// TIA Portal V19 export
DATA_BLOCK "ALARM DB PLC 2"   // DB37
{ S7_Optimized_Access := 'FALSE' }
   VAR
      "P-201 A RO 1 FEED PUMP TRIP" : Bool;
      "P-201 B RO 1 FEED PUMP TRIP" : Bool;
      "P-201 C RO 1 FEED PUMP TRIP" : Bool;
      "P-301 A RO 1 HPP PUMP TRIP" : Bool;
      "P-301 B RO B HPP PUMP TRIP" : Bool;
      "P-401 A RO 2 FEED PUMP TRIP" : Bool;
      "P-401 B RO 2 FEED PUMP TRIP" : Bool;
      "P-401 C RO 2 FEED PUMP TRIP" : Bool;
      "P 401 A RO 2 HPP PUMP TRIP" : Bool;
      "P-401 B RO 2 HPP PUMP TRIP" : Bool;
      "P-501 A EDI FEED PUMP TRIP" : Bool;
      "P-501 B EDI FEED PUMP TRIP" : Bool;
      "P-501 C EDI FEED PUMP TRIP" : Bool;
      "EDI 501 A TRIP" : Bool;
      "EDI 501 B TRIP" : Bool;
      "P-201 A RO 1 FEED PUMP_FEEDBACK FAIL" : Bool;
      "P-201 B RO 1 FEED PUMP_FEEDBACK FAIL" : Bool;
      "P-201 C RO 1 FEED PUMP_FEEDBACK FAIL" : Bool;
      "P-301 A RO 1 HPP PUMP_FEEDBACK FAIL" : Bool;
      "P-301 B RO B HPP PUMP_FEEDBACK FAIL" : Bool;
      "P-401 A RO 2 FEED PUMP_FEEDBACK FAIL" : Bool;
      "P-401 B RO 2 FEED PUMP_FEEDBACK FAIL" : Bool;
      "P-401 C RO 2 FEED PUMP_FEEDBACK FAIL" : Bool;
      "P 401 A RO 2 HPP PUMP_FEEDBACK FAIL" : Bool;
      "P-401 B RO 2 HPP PUMP_FEEDBACK FAIL" : Bool;
      "P-501 A EDI FEED PUMP_FEEDBACK FAIL" : Bool;
      "P-501 B EDI FEED PUMP_FEEDBACK FAIL" : Bool;
      "P-501 C EDI FEED PUMP_FEEDBACK FAIL" : Bool;
      "EDI 501 A _FEEDBACK FAIL" : Bool;
      "EDI 501 B_FEEDBACK FAIL" : Bool;
      "RO-01 ORP DUMP VALVE ABV-301 OPEN COMMOND FAIL" : Bool;
      "RO-01 ORP DUMP VALVE ABV-301 CLOSE COMMOND FAIL" : Bool;
      "RO-01 ORP PROCESS VALVE ABV-302 OPEN COMMOND FAIL" : Bool;
      "RO-01 ORP PROCESS VALVE ABV-302 CLOSE COMMOND FAIL" : Bool;
      "RO-1 A AUTO FLUSING VALVE AGLV-301 OPEN COMMOND FAIL" : Bool;
      "RO-1 A AUTO FLUSING VALVE AGLV-301 CLOSE COMMOND FAIL" : Bool;
      "RO-1 B AUTO FLUSING VALVE AGLV-302 OPEN COMMOND FAIL" : Bool;
      "RO-1 B AUTO FLUSING VALVE AGLV-302 CLOSE COMMOND FAIL" : Bool;
      "RO-2 A AUTO FLUSING VALVE AGLV-401 OPEN COMMOND FAIL" : Bool;
      "RO-2 A AUTO FLUSING VALVE AGLV-401 CLOSE COMMOND FAIL" : Bool;
      "RO-2 B AUTO FLUSING VALVE AGLV-402 OPEN COMMOND FAIL" : Bool;
      "RO-2 B AUTO FLUSING VALVE AGLV-402 CLOSE COMMOND FAIL" : Bool;
      "EDI AUTO DUMP VALVE ABV-501 OPEN COMMOND FAIL" : Bool;
      "EDI AUTO DUMP VALVE ABV-501 CLOSE COMMOND FAIL" : Bool;
      "DM TANK INLET VALVE ABV-502 OPEN COMMOND FAIL" : Bool;
      "DM TANK INLET VALVE ABV-502 CLOSE COMMOND FAIL" : Bool;
      "RO-02 FEED TANK LEVEL ( LT-401)- LOW LOW" : Bool;
      "RO-02 FEED TANK LEVEL ( LT-401)- HIGH HIGH" : Bool;
      "EDI FEED TANK LEVEL ( LT-501)- LOW LOW" : Bool;
      "EDI FEED TANK LEVEL ( LT-501)- HIGH HIGH" : Bool;
      "DM WATER STORAGE TANK  LEVEL ( LT-502)- LOW LOW" : Bool;
      "DM WATER STORAGE TANK LEVEL ( LT-502)- HIGH HIGH" : Bool;
      "RO-01A LPS-301 LOW" : Bool;
      "RO-01 B LPS-302 LOW" : Bool;
      "RO-01 A HPS-301 HIGH" : Bool;
      "RO-01B HPS-302 HIGH" : Bool;
      "RO-02A LPS-401 LOW" : Bool;
      "RO-02B LPS-402 LOW" : Bool;
      "RO-02A HPS-401 HIGH" : Bool;
      "RO-02 B HPS-402 HIGH" : Bool;
      "EDI-501A FEED PRESSURE PT-501 LOW" : Bool;
      "PT-501A LOW_SET VALIDATION TIME OVER_(SYSTEM STOP)" : Bool;
      "EDI-501A FEED PRESSURE PT-501 HIGH" : Bool;
      "PT-501A HIGH_SET VALIDATION TIME OVER_(SYSTEM STOP)" : Bool;
      "EDI-501B FEED PRESSURE PT-502 LOW" : Bool;
      "PT-501B LOW_SET VALIDATION TIME OVER_(SYSTEM STOP)" : Bool;
      "EDI-501B FEED PRESSURE PT-502 HIGH" : Bool;
      "PT-501B HIGH_SET VALIDATION TIME OVER_(SYSTEM STOP)" : Bool;
      "EDI-501B CONCENTRATE OUT PRESSURE PT-503 HIGH" : Bool;
      "PT-503 HIGH_SET VALIDATION TIME OVER_(SYSTEM STOP)" : Bool;
      "EDI-501A PRODUCT OUT PRESSURE PT-504 HIGH" : Bool;
      "PT-504 HIGH_SET VALIDATION TIME OVER_(SYSTEM STOP)" : Bool;
      "EDI-501A CONCENTRATE OUT PRESSURE PT-505 HIGH" : Bool;
      "PT-505 HIGH_SET VALIDATION TIME OVER_(SYSTEM STOP)" : Bool;
      "EDI-501B PRODUCT OUT PRESSURE PT-506 HIGH" : Bool;
      "PT-506 HIGH_SET VALIDATION TIME OVER_(SYSTEM STOP)" : Bool;
      "RO-01 FEED PHIT-301 HIGH" : Bool;
      "RO-01 FEED PHIT-301 LOW" : Bool;
      "RO-01 PRODUCT PHIT-302 HIGH" : Bool;
      "RO-01 PRODUCT PHIT-302 LOW" : Bool;
      "RO-02 FEED PHIT-401 HIGH" : Bool;
      "RO-02 FEED PHIT-401 LOW" : Bool;
      "RO-02 PRODUCT PHIT-402 HIGH" : Bool;
      "RO-02 PRODUCT PHIT-402 LOW" : Bool;
      "EDI-501A PRODUCT OUT  PHIT-501 HIGH" : Bool;
      "EDI-501A PRODUCT OUT  PHIT-501 LOW" : Bool;
      "EDI-501B PRODUCT OUT  PHIT-502 HIGH" : Bool;
      "EDI-501B PRODUCT OUT PHIT-502 LOW" : Bool;
      "RO-01 FEED CIT-301 HIGH" : Bool;
      "CIT-301 HIGH_SET VALIDATION TIME OVER_(SYSTEM STOP)" : Bool;
      "RO-01 PRODUCT CIT-302 HIGH" : Bool;
      "CIT-302 HIGH_SET VALIDATION TIME OVER_(SYSTEM STOP)" : Bool;
      "RO-02 FEED CIT-401 HIGH" : Bool;
      "CIT-401 HIGH_SET VALIDATION TIME OVER_(SYSTEM STOP)" : Bool;
      "RO-02 PRODUCT CIT-402 HIGH" : Bool;
      "CIT-402 HIGH_SET VALIDATION TIME OVER_(SYSTEM STOP)" : Bool;
      "EDI-501A PRODUCT OUT RIT-501 HIGH" : Bool;
      "RIT-501A HIGH_SET VALIDATION TIME OVER_(SYSTEM STOP)" : Bool;
      "EDI-501B PRODUCT OUT RIT-502 HIGH" : Bool;
      "RIT-501B HIGH_SET VALIDATION TIME OVER_(SYSTEM STOP)" : Bool;
      "ORP-301 HIGH" : Bool;
      "ORP-301 HIGH_SET VALIDATION TIME OVER_(SYSTEM STOP)" : Bool;
      "EDI-501A FEED PRESSURE FIT-501 LOW" : Bool;
      "FIT-501  LOW_SET VALIDATION TIME OVER_(SYSTEM STOP)" : Bool;
      "EDI-501B FEED PRESSURE FIT-502 LOW" : Bool;
      "FIT-501 LOW_SET VALIDATION TIME OVER_(SYSTEM STOP)" : Bool;
      "EDI-501B CONCENTRATE OUT PRESSURE FIT-503 LOW" : Bool;
      "FIT-503 LOW_SET VALIDATION TIME OVER_(SYSTEM STOP)" : Bool;
      "EDI-501A PRODUCT OUT PRESSURE FIT-504 LOW" : Bool;
      "FIT-504 LOW_SET VALIDATION TIME OVER_(SYSTEM STOP)" : Bool;
      "EDI-501B CONCENTRATE OUT PRESSURE FIT-505 LOW" : Bool;
      "FIT-505 LOW_SET VALIDATION TIME OVER_(SYSTEM STOP)" : Bool;
      "EDI-501B CONCENTRATE OUT PRESSURE FIT-505 HIGH" : Bool;
      "FIT-505 HIGH_SET VALIDATION TIME OVER_(SYSTEM STOP)" : Bool;
      "EDI-501A PRODUCT OUT PRESSURE FIT-506 LOW" : Bool;
      "FIT-506 LOW_SET VALIDATION TIME OVER_(SYSTEM STOP)" : Bool;
      "EDI-501A PRODUCT OUT PRESSURE FIT-506 HIGH" : Bool;
      "FIT-506 HIGH_SET VALIDATION TIME OVER_(SYSTEM STOP)" : Bool;
      "EDI-501B CONCENTRATE OUT PRESSURE FIT-507 LOW" : Bool;
      "FIT-507 LOW_SET VALIDATION TIME OVER_(SYSTEM STOP)" : Bool;
      "EDI-501B CONCENTRATE OUT PRESSURE FIT-507 HIGH" : Bool;
      "FIT-507 HIGH_SET VALIDATION TIME OVER_(SYSTEM STOP)" : Bool;
      "EDI-501A PRODUCT OUT PRESSURE FIT-508 LOW" : Bool;
      "FIT-508 LOW_SET VALIDATION TIME OVER_(SYSTEM STOP)" : Bool;
      "EDI-501A PRODUCT OUT PRESSURE FIT-508 HIGH" : Bool;
      "FIT-508 HIGH_SET VALIDATION TIME OVER_(SYSTEM STOP)" : Bool;
   END_VAR
BEGIN
END_DATA_BLOCK
